Omron CX-Programmer project NewProject (CX-Programmer 9.75)

# PLC NewPLC1: CP1L M

## Global symbols (name address type ; comment)
test _INV201_ReadParameter

## Program NewProgram1 (cyclic task 0)

### Section Section1

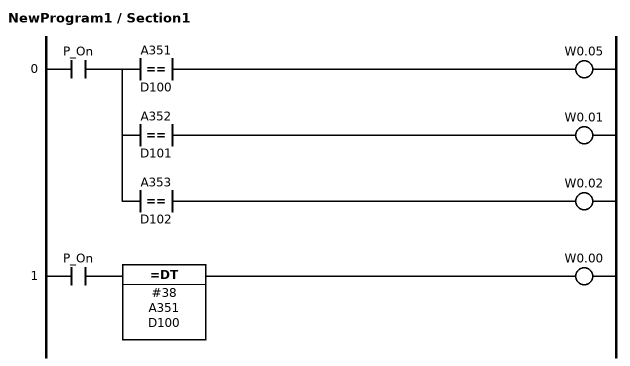
; rung 0
LD P_On
OUT TR0
AND=(300) A351 D100
OUT W0.05
LD TR0
AND=(300) A352 D101
OUT W0.01
LD TR0
AND=(300) A353 D102
OUT W0.02
; rung 1
LD P_On
AND=DT(341) #38 A351 D100
OUT W0.00

### Section END
; rung 0
END(001)

## Function block _INV201_ReadParameter (Omron library block, body left out)